{attribute 'GeneratedUsingTerminal: IODEVICETYPE_ETHERCATPROT'}
{attribute addProperty BoxType "IODEVICETYPE_ETHERCATPROT"}
{attribute addProperty Id "Beckhoff_ELM3xxxBeckhoff_ELM3xxx_EC7DF201384Beckhoff_ELM31xxBeckhoff_ELM31xx_6C09EABC1114Beckhoff_ELM35xxBeckhoff_ELM35xx_F2A46C7A426Beckhoff_ELM36xxBeckhoff_ELM36xx_F21F91D5532Beckhoff_ELM37xxBeckhoff_ELM37xx_58029B3E512Beckhoff_ELM3xxx_0030Beckhoff_ELM3xxx_0030_4ED1F717320Beckhoff_ELM9xxxBeckhoff_ELM9xxx_4C94887B367SyncUnitsSyncUnits_99E584AF18InputsInputs_25A0042B160OutputsOutputs_2397A10E106InfoDataInfoData_C76BEFB322"}
{attribute addProperty CRC "4259140306"}
{attribute addProperty Size "3961"}
TYPE EtherCAT_Master_ELMxxxx_FDDD52D2 :
STRUCT
	{attribute addProperty Name "Beckhoff_ELM3xxx"}
	{attribute addProperty PreviousPort "EtherCAT_Master_ELMxxxx : Master"}
	Beckhoff_ELM3xxx : Beckhoff_ELM3xxx_EC7DF201;
	{attribute addProperty Name "Beckhoff_ELM31xx"}
	{attribute addProperty PreviousPort "Beckhoff ELM3xxx : C"}
	Beckhoff_ELM31xx : Beckhoff_ELM31xx_6C09EABC;
	{attribute addProperty Name "Beckhoff_ELM35xx"}
	{attribute addProperty PreviousPort "Beckhoff ELM31xx : C"}
	Beckhoff_ELM35xx : Beckhoff_ELM35xx_F2A46C7A;
	{attribute addProperty Name "Beckhoff_ELM36xx"}
	{attribute addProperty PreviousPort "Beckhoff ELM35xx : C"}
	Beckhoff_ELM36xx : Beckhoff_ELM36xx_F21F91D5;
	{attribute addProperty Name "Beckhoff_ELM37xx"}
	{attribute addProperty PreviousPort "Beckhoff ELM36xx : C"}
	Beckhoff_ELM37xx : Beckhoff_ELM37xx_58029B3E;
	{attribute addProperty Name "Beckhoff_ELM3xxx_0030"}
	{attribute addProperty PreviousPort "Beckhoff ELM37xx : C"}
	Beckhoff_ELM3xxx_0030 : Beckhoff_ELM3xxx_0030_4ED1F717;
	{attribute addProperty Name "Beckhoff_ELM9xxx"}
	{attribute addProperty PreviousPort "Beckhoff ELM3xxx-0030 : C"}
	Beckhoff_ELM9xxx : Beckhoff_ELM9xxx_4C94887B;
	{attribute addProperty Name "SyncUnits"}
	SyncUnits : SyncUnits_99E584AF;
	{attribute addProperty Name "Inputs"}
	Inputs : Inputs_25A0042B;
	{attribute addProperty Name "Outputs"}
	Outputs : Outputs_2397A10E;
	{attribute addProperty Name "InfoData"}
	InfoData : InfoData_C76BEFB3;
END_STRUCT
END_TYPE

(* stored: Version 1.2.0.0, ProductVersion 3.1.4024.9
   DUT EtherCAT_Master_ELMxxxx_FDDD52D2: Id {3c55207e-fa74-4239-bd38-eba55b3700ac} *)
